// TIA Portal V17 export
// export: Created 2026-04-13T11:12:42.157199Z, ExportSetting WithDefaults, DisplayName Totally Integrated Automation Portal, DisplayVersion V17 Update 4, DisplayName TIA Portal Openness, DisplayVersion V17 Update 4, DisplayName TIA Portal Version Control Interface, DisplayVersion V17, DisplayName SINAMICS Startdrive Advanced, DisplayVersion V17, DisplayName SINAMICS Startdrive G130, G150, S120, S150, SINAMICS MV, S210, DisplayVersion V17, DisplayName SINAMICS Startdrive G110M, G120, G120C, G120D, G120P, G115D, DisplayVersion V17, DisplayName STEP 7 Professional, DisplayVersion V17 Update 4, DisplayName STEP 7 Safety, DisplayVersion V17, DisplayName WinCC Professional, DisplayVersion V17 Update 4
FUNCTION_BLOCK "沿"   // FB67, LAD
{ S7_Optimized_Access := 'TRUE' }
VERSION : 0.1
// stored: AutoNumber true, IsIECCheckEnabled false, IsRetainMemResEnabled false, MemoryReserve 100, SetENOAutomatically false, UDAEnableTagReadback false
   VAR_INPUT
      IN : Bool;
   END_VAR
   VAR_OUTPUT
      Q : Bool;
   END_VAR
   VAR
      U_1 : Bool;
      L_1 : Bool;
   END_VAR
BEGIN

REGION Network 1 (SCL)
   IF #IN AND NOT #U_1 THEN

       #Q := 1;

   END_IF;

   #U_1 := #IN;
END_REGION
END_FUNCTION_BLOCK
